// TIA Portal V15 export
// export: Created 2019-02-22T09:02:27.6652563Z, ExportSetting WithDefaults, WithReadOnly, DisplayName Totally Integrated Automation Portal, DisplayVersion V15 Update 2, DisplayName TIA Portal Openness, DisplayVersion V15 Update 2, DisplayName STEP 7 Professional, DisplayVersion V15 Update 2, DisplayName STEP 7 Safety, DisplayVersion V15, DisplayName WinCC Professional, DisplayVersion V15 Update 2, DisplayName SIMATIC Visualization Architect, DisplayVersion V15 Update 1
FUNCTION "STATION_NAME_Call" : Void   // FC10, FBD
TITLE = Call STATION_NAME / Station STATION_NAME
{ S7_Optimized_Access := 'FALSE' }
VERSION : 0.1
// stored: AutoNumber true, CodeModifiedDate 2019-01-06T16:26:05.7067541Z, CompileDate 2019-01-06T16:26:05.7918278Z, CreationDate 2018-11-16T09:32:53.5033139Z, HandleErrorsWithinBlock false, InterfaceModifiedDate 2016-02-03T14:10:26.7352599Z, IsConsistent true, IsIECCheckEnabled false, IsKnowHowProtected false, IsWriteProtected false, LibraryConformanceStatus Error: The block contains calls of single instances. Warning: The object contains access to global data blocks. Warning: The block contains direct access to inputs, outputs, bit memories, indirect access to the registry or indirect access to external memory areas that are unknown at the time of compilation., ModifiedDate 2019-01-06T16:26:05.7067541Z, ParameterModified 2016-02-03T14:10:26.7196349Z, PLCSimAdvancedSupport true, SetENOAutomatically False, StructureModified 2016-02-03T14:10:26.7352599Z, UDAEnableTagReadback false
   VAR_TEMP   // added for the SCL form of the ladder/FBD networks
      _w1 : Bool;
   END_VAR
BEGIN

REGION Network 1: Grundstellung
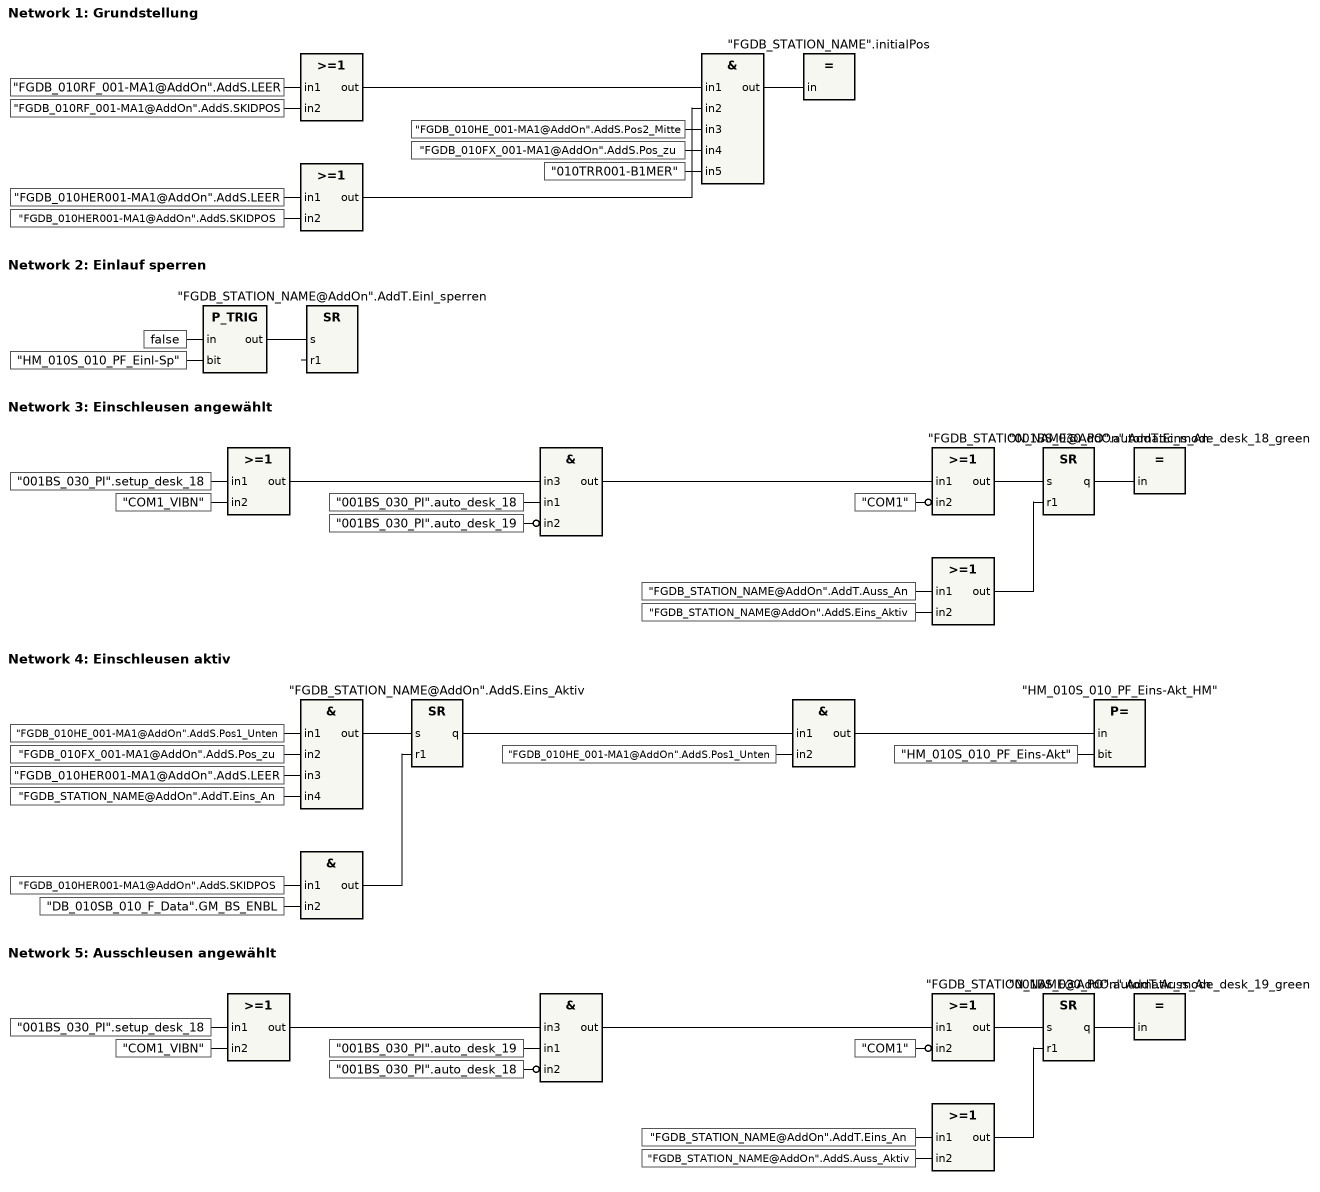
   "FGDB_STATION_NAME".initialPos := ("FGDB_010RF_001-MA1@AddOn".AddS.LEER OR "FGDB_010RF_001-MA1@AddOn".AddS.SKIDPOS) AND ("FGDB_010HER001-MA1@AddOn".AddS.LEER OR "FGDB_010HER001-MA1@AddOn".AddS.SKIDPOS) AND "FGDB_010HE_001-MA1@AddOn".AddS.Pos2_Mitte AND "FGDB_010FX_001-MA1@AddOn".AddS.Pos_zu AND "010TRR001-B1MER";
END_REGION

REGION Network 2: Einlauf sperren
   #_w1 := false AND NOT "HM_010S_010_PF_Einl-Sp";   // rising edge
   "HM_010S_010_PF_Einl-Sp" := false;
   IF #_w1 THEN
       "FGDB_STATION_NAME@AddOn".AddT.Einl_sperren := TRUE;   // SR flip-flop
   END_IF;
END_REGION

REGION Network 3: Einschleusen angewählt
   // 1. auto_desk_18 = Taster Einschleusen
   // 2. setup_desk_18_ Taster Frg. Übernehmen
   // 3. auto_desk_19 = Taster Ausschleusen
   IF (("001BS_030_PI".setup_desk_18 OR "COM1_VIBN") AND "001BS_030_PI".auto_desk_18 AND NOT "001BS_030_PI".auto_desk_19) OR NOT "COM1" THEN
       "FGDB_STATION_NAME@AddOn".AddT.Eins_An := TRUE;   // SR flip-flop
   END_IF;
   IF "FGDB_STATION_NAME@AddOn".AddT.Auss_An OR "FGDB_STATION_NAME@AddOn".AddS.Eins_Aktiv THEN
       "FGDB_STATION_NAME@AddOn".AddT.Eins_An := FALSE;
   END_IF;
   "001BS_030_PO".automatic_mode_desk_18_green := "FGDB_STATION_NAME@AddOn".AddT.Eins_An;
END_REGION

REGION Network 4: Einschleusen aktiv
   IF "FGDB_010HE_001-MA1@AddOn".AddS.Pos1_Unten AND "FGDB_010FX_001-MA1@AddOn".AddS.Pos_zu AND "FGDB_010HER001-MA1@AddOn".AddS.LEER AND "FGDB_STATION_NAME@AddOn".AddT.Eins_An THEN
       "FGDB_STATION_NAME@AddOn".AddS.Eins_Aktiv := TRUE;   // SR flip-flop
   END_IF;
   IF "FGDB_010HER001-MA1@AddOn".AddS.SKIDPOS AND "DB_010SB_010_F_Data".GM_BS_ENBL THEN
       "FGDB_STATION_NAME@AddOn".AddS.Eins_Aktiv := FALSE;
   END_IF;
   #_w1 := "FGDB_STATION_NAME@AddOn".AddS.Eins_Aktiv AND "FGDB_010HE_001-MA1@AddOn".AddS.Pos1_Unten;
   "HM_010S_010_PF_Eins-Akt_HM" := #_w1 AND NOT "HM_010S_010_PF_Eins-Akt";   // rising edge
   "HM_010S_010_PF_Eins-Akt" := #_w1;
END_REGION

REGION Network 5: Ausschleusen angewählt
   // 1. auto_desk_18 = Taster Einschleusen
   // 2. setup_desk_18_ Taster Frg. Übernehmen
   // 3. auto_desk_19 = Taster Ausschleusen
   IF (("001BS_030_PI".setup_desk_18 OR "COM1_VIBN") AND "001BS_030_PI".auto_desk_19 AND NOT "001BS_030_PI".auto_desk_18) OR NOT "COM1" THEN
       "FGDB_STATION_NAME@AddOn".AddT.Auss_An := TRUE;   // SR flip-flop
   END_IF;
   IF "FGDB_STATION_NAME@AddOn".AddT.Eins_An OR "FGDB_STATION_NAME@AddOn".AddS.Auss_Aktiv THEN
       "FGDB_STATION_NAME@AddOn".AddT.Auss_An := FALSE;
   END_IF;
   "001BS_030_PO".automatic_mode_desk_19_green := "FGDB_STATION_NAME@AddOn".AddT.Auss_An;
END_REGION

REGION Network 6: Ausschleusen aktiv
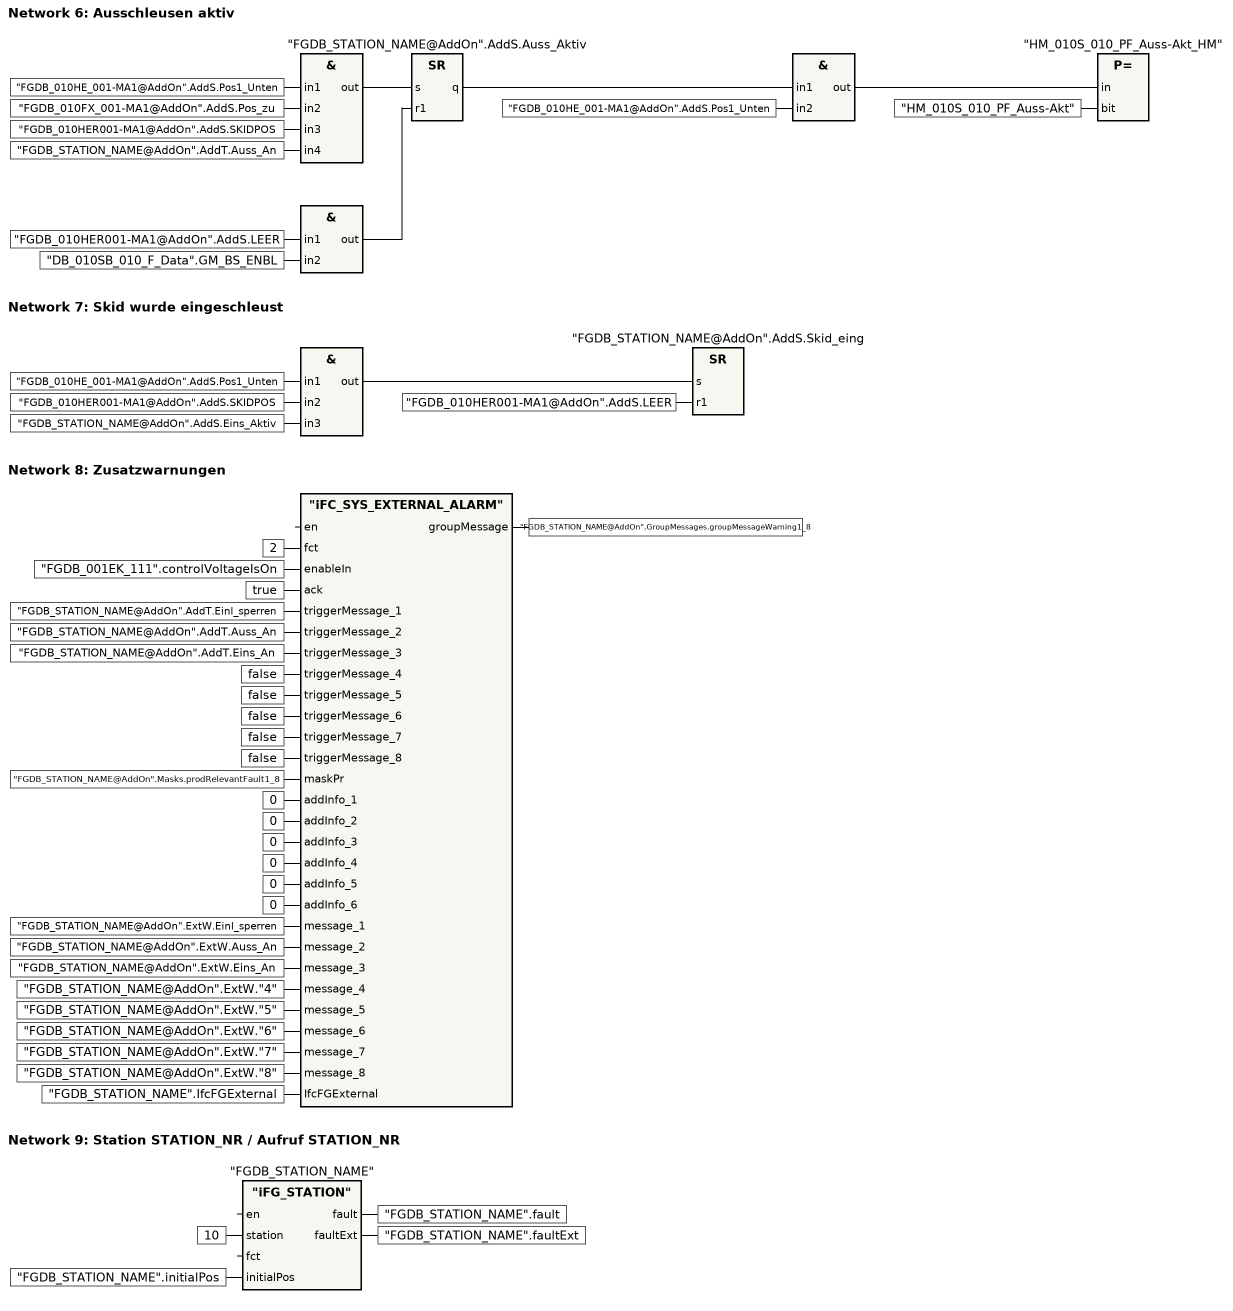
   IF "FGDB_010HE_001-MA1@AddOn".AddS.Pos1_Unten AND "FGDB_010FX_001-MA1@AddOn".AddS.Pos_zu AND "FGDB_010HER001-MA1@AddOn".AddS.SKIDPOS AND "FGDB_STATION_NAME@AddOn".AddT.Auss_An THEN
       "FGDB_STATION_NAME@AddOn".AddS.Auss_Aktiv := TRUE;   // SR flip-flop
   END_IF;
   IF "FGDB_010HER001-MA1@AddOn".AddS.LEER AND "DB_010SB_010_F_Data".GM_BS_ENBL THEN
       "FGDB_STATION_NAME@AddOn".AddS.Auss_Aktiv := FALSE;
   END_IF;
   #_w1 := "FGDB_STATION_NAME@AddOn".AddS.Auss_Aktiv AND "FGDB_010HE_001-MA1@AddOn".AddS.Pos1_Unten;
   "HM_010S_010_PF_Auss-Akt_HM" := #_w1 AND NOT "HM_010S_010_PF_Auss-Akt";   // rising edge
   "HM_010S_010_PF_Auss-Akt" := #_w1;
END_REGION

REGION Network 7: Skid wurde eingeschleust
   IF "FGDB_010HE_001-MA1@AddOn".AddS.Pos1_Unten AND "FGDB_010HER001-MA1@AddOn".AddS.SKIDPOS AND "FGDB_STATION_NAME@AddOn".AddS.Eins_Aktiv THEN
       "FGDB_STATION_NAME@AddOn".AddS.Skid_eing := TRUE;   // SR flip-flop
   END_IF;
   IF "FGDB_010HER001-MA1@AddOn".AddS.LEER THEN "FGDB_STATION_NAME@AddOn".AddS.Skid_eing := FALSE; END_IF;
END_REGION

REGION Network 8: Zusatzwarnungen
   "iFC_SYS_EXTERNAL_ALARM"(fct := 2,
                           enableIn := "FGDB_001EK_111".controlVoltageIsOn,
                           ack := true,
                           triggerMessage_1 := "FGDB_STATION_NAME@AddOn".AddT.Einl_sperren,
                           triggerMessage_2 := "FGDB_STATION_NAME@AddOn".AddT.Auss_An,
                           triggerMessage_3 := "FGDB_STATION_NAME@AddOn".AddT.Eins_An,
                           triggerMessage_4 := false,
                           triggerMessage_5 := false,
                           triggerMessage_6 := false,
                           triggerMessage_7 := false,
                           triggerMessage_8 := false,
                           maskPr := "FGDB_STATION_NAME@AddOn".Masks.prodRelevantFault1_8,
                           addInfo_1 := 0,
                           addInfo_2 := 0,
                           addInfo_3 := 0,
                           addInfo_4 := 0,
                           addInfo_5 := 0,
                           addInfo_6 := 0,
                           message_1 := "FGDB_STATION_NAME@AddOn".ExtW.Einl_sperren,
                           message_2 := "FGDB_STATION_NAME@AddOn".ExtW.Auss_An,
                           message_3 := "FGDB_STATION_NAME@AddOn".ExtW.Eins_An,
                           message_4 := "FGDB_STATION_NAME@AddOn".ExtW."4",
                           message_5 := "FGDB_STATION_NAME@AddOn".ExtW."5",
                           message_6 := "FGDB_STATION_NAME@AddOn".ExtW."6",
                           message_7 := "FGDB_STATION_NAME@AddOn".ExtW."7",
                           message_8 := "FGDB_STATION_NAME@AddOn".ExtW."8",
                           IfcFGExternal := "FGDB_STATION_NAME".IfcFGExternal,
                           groupMessage => "FGDB_STATION_NAME@AddOn".GroupMessages.groupMessageWarning1_8);
END_REGION

REGION Network 9: Station STATION_NR / Aufruf STATION_NR
   "FGDB_STATION_NAME"(station := 10,   // "iFG_STATION"
                       initialPos := "FGDB_STATION_NAME".initialPos,
                       fault => "FGDB_STATION_NAME".fault,
                       faultExt => "FGDB_STATION_NAME".faultExt);
END_REGION
END_FUNCTION
